{attribute 'hide'}
FUNCTION INTERNAL FormatString2 : T_MaxString
VAR_INPUT
	Format	: T_MaxString;
	arg1	: T_Arg;
	arg2	: T_Arg;
END_VAR
VAR
    FB_FormatString1 : FB_FormatString;
END_VAR

FB_FormatString1(sFormat := Format,
                 arg1    := arg1,
                 arg2    := arg2,
                 arg3    :=,
                 arg4    :=,
                 arg5    :=,
                 arg6    :=,
                 arg7    :=,
                 arg8    :=,
                 arg9    :=,
                 arg10   :=,
                 bError  =>,
                 nErrId  =>,
                 sOut    => FormatString2);

END_FUNCTION

(* stored: Version 1.1.0.1, ProductVersion 3.1.4024.12
   POU FormatString2: Id {8c150b92-44dc-0568-210b-eedfde30141b}, SpecialFunc None *)
